// TIA Portal V20 export
VAR_GLOBAL   // PLC tag table "Standard"
   false AT %M0.0 : Bool;
   true AT %M0.1 : Bool;
   test0 AT %M0.2 : Bool;
   test1 AT %M0.3 : Bool;
   dummy AT %M0.7 : Bool;
   clockFlag10Hz AT %M1.0 : Bool;   // ClockFlag 0.1s
   clockFlag5Hz AT %M1.1 : Bool;   // ClockFlag 0.2s
   flash AT %M1.2 : Bool;   // ClockFlag 0.4s
   clockFlag2Hz AT %M1.3 : Bool;   // ClockFlag 0.5s
   blinker AT %M1.4 : Bool;   // ClockFlag 0.8s
   clockFlag1Hz AT %M1.5 : Bool;   // ClockFlag 1.0s
   "clockFlag0,625Hz" AT %M1.6 : Bool;   // ClockFlag 1.6s
   "clockFlag0,5Hz" AT %M1.7 : Bool;   // ClockFlag 2.0s
   cycleFlag AT %MB2 : Byte;
   cycleFlash AT %M2.0 : Bool;
   systemByte AT %MB3 : Byte;
   firstScan AT %M3.0 : Bool;   // cpu startup
   diagStatusUpdate AT %M3.1 : Bool;
   alwaysTRUE AT %M3.2 : Bool;
   alwaysFALSE AT %M3.3 : Bool;
   clockByte AT %MB1 : Byte;
   cycle AT %MD6 : Real;   // program cycle in ms
   "real" AT %MD10 : Real;
   "dWord" AT %MD18 : DWord;
   "dint" AT %MD14 : DInt;
   "int" AT %MW22 : Int;
   "word" AT %MW24 : Word;
   "byte" AT %MB26 : Byte;
   "bool" AT %M27.0 : Bool;
   systemClockByte AT %MB30 : Byte;
   clockTest AT %M0.6 : Bool;
   T0 AT %T0 : Timer;
   T1 AT %T1 : Timer;
   T2 AT %T2 : Timer;
   mem AT %M32.0 : LReal;
   T3 AT %T3 : Timer;
END_VAR
